FUNCTION_BLOCK FB_Arguments IMPLEMENTS Tc3_EventLogger.I_TcArguments
VAR_INPUT
	sOriginalString:		STRING(255);
	iInterfacePointer:		Tc3_EventLogger.I_TcArguments;
END_VAR
VAR_OUTPUT
	sOutText:				STRING(255);
END_VAR
VAR
	ipArgumentsinterface:	Tc3_EventLogger.I_TcArguments;
	bInit: 					BOOL := TRUE;
END_VAR

IF			bInit THEN
	bInit := FALSE;
	Clear();
END_IF

METHOD AddBlob : Tc3_EventLogger.I_TcArguments
VAR_INPUT
	pData	: Tc3_EventLogger.PVOID;
	cbData	: UINT;
END_VAR
END_METHOD

METHOD AddBool : Tc3_EventLogger.I_TcArguments
VAR_INPUT
	value	: BOOL;
END_VAR
VAR
	sValue:	STRING;
END_VAR
sValue := BOOL_TO_STRING(value);
AddString(sValue);
AddBool := iInterfacePointer;
END_METHOD

METHOD AddByte : Tc3_EventLogger.I_TcArguments
VAR_INPUT
	value	: BYTE;
END_VAR
VAR
	sValue:	STRING;
END_VAR
sValue := (BYTE_TO_STRING(value));
AddString(sValue);
AddByte := iInterfacePointer;
END_METHOD

METHOD AddDInt : Tc3_EventLogger.I_TcArguments
VAR_INPUT
	value	: DINT;
END_VAR
VAR
	sValue:	STRING;
END_VAR
sValue := (DINT_TO_STRING(value));
AddString(sValue);
AddDInt := iInterfacePointer;
END_METHOD

METHOD AddDWord : Tc3_EventLogger.I_TcArguments
VAR_INPUT
	value	: DWORD;
END_VAR
VAR
	sValue:	STRING;
END_VAR
sValue := (DWORD_TO_STRING(value));
AddString(sValue);
AddDWord := iInterfacePointer;
END_METHOD

METHOD AddEventReferenceEx : Tc3_EventLogger.I_TcArguments
VAR_INPUT
	stEventEntry	: Tc3_EventLogger.TcEventEntry;
END_VAR
END_METHOD

METHOD AddEventReferenceId : Tc3_EventLogger.I_TcArguments
VAR_INPUT
	nEventId	: UDINT;
END_VAR
END_METHOD

METHOD AddEventReferenceIdGuid : Tc3_EventLogger.I_TcArguments
VAR_INPUT
	nEventId	: UDINT;
	EventClass	: Tc3_EventLogger.GUID;
END_VAR
END_METHOD

METHOD AddInt : Tc3_EventLogger.I_TcArguments
VAR_INPUT
	value	: INT;
END_VAR
VAR
	sValue:	STRING;
END_VAR
sValue := (INT_TO_STRING(value));
AddString(sValue);
AddInt := iInterfacePointer;
END_METHOD

METHOD AddLInt : Tc3_EventLogger.I_TcArguments
VAR_INPUT
	value	: LINT;
END_VAR
VAR
	sValue:	STRING;
END_VAR
sValue := (LINT_TO_STRING(value));
AddString(sValue);
AddLInt := iInterfacePointer;
END_METHOD

METHOD AddLReal : Tc3_EventLogger.I_TcArguments
VAR_INPUT
	value	: LREAL;
END_VAR
VAR
	sValue:	STRING;
END_VAR
sValue := (LREAL_TO_STRING(value));
AddString(sValue);
AddLReal := iInterfacePointer;
END_METHOD

METHOD AddReal : Tc3_EventLogger.I_TcArguments
VAR_INPUT
	value	: REAL;
END_VAR
VAR
	sValue:	STRING;
END_VAR
sValue := (REAL_TO_STRING(value));
AddString(sValue);
AddReal := iInterfacePointer;
END_METHOD

METHOD AddSInt : Tc3_EventLogger.I_TcArguments
VAR_INPUT
	value	: SINT;
END_VAR
VAR
	sValue:	STRING;
END_VAR
sValue := (SINT_TO_STRING(value));
AddString(sValue);
AddSInt := iInterfacePointer;
END_METHOD

METHOD AddString : Tc3_EventLogger.I_TcArguments
VAR_IN_OUT CONSTANT
	value	: STRING;
END_VAR
VAR
	nPosition:		INT;
END_VAR
nPosition := getNextPlaceholder();
IF			(nPosition > 0) THEN
	sOutText := INSERT(Delete(sOutText, 3, nPosition), value, nPosition-1);
END_IF

AddString := iInterfacePointer;
END_METHOD

METHOD AddStringByValue : Tc3_EventLogger.I_TcArguments
VAR_INPUT
	value	: Tc3_EventLogger.T_MaxString;
END_VAR
END_METHOD

METHOD AddUDInt : Tc3_EventLogger.I_TcArguments
VAR_INPUT
	value	: UDINT;
END_VAR
VAR
	sValue:	STRING;
END_VAR
sValue := (UDINT_TO_STRING(value));
AddString(sValue);
AddUDInt := iInterfacePointer;
END_METHOD

METHOD AddUInt : Tc3_EventLogger.I_TcArguments
VAR_INPUT
	value	: UINT;
END_VAR
VAR
	sValue:	STRING;
END_VAR
sValue := (UINT_TO_STRING(value));
AddString(sValue);
AddUInt := iInterfacePointer;
END_METHOD

METHOD AddULInt : Tc3_EventLogger.I_TcArguments
VAR_INPUT
	value	: ULINT;
END_VAR
VAR
	sValue:	STRING;
END_VAR
sValue := (ULINT_TO_STRING(value));
AddString(sValue);
AddULInt := iInterfacePointer;
END_METHOD

METHOD AddUSInt : Tc3_EventLogger.I_TcArguments
VAR_INPUT
	value	: USINT;
END_VAR
VAR
	sValue:	STRING;
END_VAR
sValue := (USINT_TO_STRING(value));
AddString(sValue);
AddUSInt := iInterfacePointer;
END_METHOD

METHOD AddUtf8EncodedString : Tc3_EventLogger.I_TcArguments
VAR_IN_OUT CONSTANT
	value	: STRING;
END_VAR
END_METHOD

METHOD AddWord : Tc3_EventLogger.I_TcArguments
VAR_INPUT
	value	: WORD;
END_VAR
VAR
	sValue:	STRING;
END_VAR
sValue := (WORD_TO_STRING(value));
AddString(sValue);
AddWord := iInterfacePointer;
END_METHOD

METHOD AddWString : Tc3_EventLogger.I_TcArguments
VAR_IN_OUT CONSTANT
	value	: WSTRING;
END_VAR
END_METHOD

METHOD AddWStringByValue : Tc3_EventLogger.I_TcArguments
VAR_INPUT
	value	: WSTRING(255);
END_VAR
END_METHOD

METHOD Clear : Tc3_EventLogger.I_TcArguments
sOutText := sOriginalString;
Clear := iInterfacePointer;
END_METHOD

METHOD getNextPlaceholder : INT
VAR_INPUT
END_VAR
VAR
	sText:					STRING(255);
	nPosition:				INT;
	nPlaceholder:			INT;
	nNextPlaceholder:		INT := 32767;
	nNextPlaceholderPos:	INT;
	
	nDeleted:				INT;
	
	bNoMorePlaceholders:	BOOL;
END_VAR
sText := sOutText;

REPEAT
	nPosition := FIND(sText, '{');
	
	IF			(nPosition > 0) THEN
		nPlaceholder := STRING_TO_INT(MID(sText, 1, nPosition+1));
		
		IF			(nPlaceholder < nNextPlaceholder) THEN
			nNextPlaceholder := nPlaceholder;
			nNextPlaceholderPos := nPosition+nDeleted;
		END_IF
		
		sText := Delete(sText, nPosition+2, 1);		//Alles bis zum Plazhalter löschen
		nDeleted := nDeleted+nPosition+2;
		
	ELSE
		bNoMorePlaceholders := TRUE;
	END_IF
	
UNTIL 
	bNoMorePlaceholders
END_REPEAT

getNextPlaceholder := nNextPlaceholderPos;
END_METHOD

PROPERTY ipData : Tc3_EventLogger.ITcArguments
GET
END_GET
END_PROPERTY

PROPERTY nCount : UDINT
GET
END_GET
END_PROPERTY

END_FUNCTION_BLOCK

(* stored: Version 1.1.0.1, ProductVersion 3.1.4024.12
   POU FB_Arguments: Id {2f4b86c3-73aa-43a3-8474-dfcdd1e32a6b}, SpecialFunc None
   Method AddBlob: Id {875da798-9b04-43b9-b2bb-cabb22622ed0}
   Method AddBool: Id {550c5e5e-51b9-4872-b477-1677f0600b2b}
   Method AddByte: Id {85534321-4a35-4332-8c4a-bfb2f277ecf2}
   Method AddDInt: Id {619ad327-6da6-47b0-860f-7b4efee6a90f}
   Method AddDWord: Id {f6f20f8b-f4ae-4b8d-93cc-8bc6a67ddf6d}
   Method AddEventReferenceEx: Id {55f7b3fe-899d-4d5c-aa68-5b29f6b3721f}
   Method AddEventReferenceId: Id {7529b9ca-c485-4827-ba9e-c4c796dfff7e}
   Method AddEventReferenceIdGuid: Id {7343f831-c2de-44b7-ab52-c0a5c43fd93d}
   Method AddInt: Id {2a79c6a0-cbf7-4cd5-ac6d-57e99e13ef9f}
   Method AddLInt: Id {5a8aad80-fb00-4047-928d-683ad9a4c514}
   Method AddLReal: Id {1a617b08-6423-4282-bfa6-893eabba7116}
   Method AddReal: Id {a863ca27-c5ef-4e76-a329-abb73f1dd5f6}
   Method AddSInt: Id {49f9be51-0e62-42e2-8033-71648ca00118}
   Method AddString: Id {67feb8ac-ed9e-4a3d-9816-2ca62643e197}
   Method AddStringByValue: Id {162ad298-68ba-4b19-999d-6862b7f56066}
   Method AddUDInt: Id {84e039a9-baa7-4733-8b4f-bb3152628288}
   Method AddUInt: Id {c334a718-914e-4d55-b26b-41cd92905ed2}
   Method AddULInt: Id {dd7f2def-fe53-4099-b8fb-249c8d9b93b6}
   Method AddUSInt: Id {162ae065-474b-4ef6-a88b-4d860af857fb}
   Method AddUtf8EncodedString: Id {54b62175-b051-46a3-92b0-5d151e61a660}
   Method AddWord: Id {73310218-f73b-4601-be6c-b60df8d4956b}
   Method AddWString: Id {8cbcabeb-001e-45d4-a01c-5ad1646542da}
   Method AddWStringByValue: Id {1c64c112-3fa0-446f-ab74-32a273522483}
   Method Clear: Id {7ab18b35-e651-4e2b-9505-0030e005715f}
   Method getNextPlaceholder: Id {25bb079a-ce4d-4632-a1cf-9b6887d170a3}
   Property ipData: Id {878d5534-4c75-4eb0-8db9-aadfd9015a47}
   Get Get: Id {d7d46211-1d8a-47d4-8fe0-600a8b3ba4d0}
   Property nCount: Id {d63fde19-71d8-4e28-bc40-c2c00481cef7}
   Get Get: Id {172dc9fa-8d70-4423-8a80-0569cae84136} *)
